FUNCTION_BLOCK FB_Infeed
VAR_INPUT
	bEnable_Master			: BOOL;
	bMoveMaster				: BOOL;
	bSensorProduct			: BOOL;
END_VAR

VAR_IN_OUT
	Master					: Axis_Ref;
	VirtMaster				: ARRAY [*] OF Axis_Ref;
END_VAR

VAR
	i						: DINT;
	iStartIndex				: DINT;
	VeloMaster				: LREAL;
	bToggle					: BOOL;

	fbPowerMaster			: MC_Power;
	fbMoveMaster			: MC_MoveVelocity;
	fbStopMaster			: MC_Halt;
	fbPowerVirtMaster		: ARRAY [1..iMaxNumbVirtMasters] OF MC_Power;
	fbVirtMaster			: ARRAY [1..iMaxNumbVirtMasters] OF FB_VirtualMaster;

END_VAR

// Enable Master
Master.ReadStatus();
fbPowerMaster(
	Axis			:= Master, 
	Enable			:= bEnable_Master, 
	Enable_Positive	:= bEnable_Master, 
	Enable_Negative	:= bEnable_Master, 
	Override		:= 100, 
	);
	
FOR i := 1 TO UPPER_BOUND(VirtMaster,1) DO
	VirtMaster[i].ReadStatus();
	fbPowerVirtMaster[i](
		Axis			:= VirtMaster[i], 
		Enable			:= bEnable_Master, 
		Enable_Positive	:= bEnable_Master, 
		Enable_Negative	:= bEnable_Master, 
		Override		:= 100, 
		);
END_FOR


// Start-Stop Master

VeloMaster := GVL_Infeed.iProductsPerMinute * 360 / 60;
bToggle:=NOT bToggle;

fbMoveMaster(
	Axis		:= Master, 
	Execute		:= bMoveMaster AND bToggle, 
	Velocity	:= VeloMaster, 
	Direction	:= MC_Positive_Direction, 
	);
fbStopMaster(
	Axis		:= Master, 
	Execute		:= NOT bMoveMaster, 
	);

// Virtual Master ready to start
iStartIndex:=0;
FOR i := 1 TO UPPER_BOUND(VirtMaster,1) DO
	IF VirtMaster[i].NcToPlc.ActPos=0 THEN
		iStartIndex:=i;
		i:=5;
	END_IF
END_FOR
	
// Detection product
FOR i := 1 TO UPPER_BOUND(VirtMaster,1) DO
	fbVirtMaster[i].bActivateCam:=FALSE;
END_FOR

IF (Master.NcToPlc.ModuloActPos > GVL_Infeed.rDetectionPosMin) AND (Master.NcToPlc.ModuloActPos < GVL_Infeed.rDetectionPosMax) AND bSensorProduct THEN
	fbVirtMaster[iStartIndex].bActivateCam:=TRUE;
END_IF
 
FOR i := 1 TO UPPER_BOUND(VirtMaster,1) DO
	fbVirtMaster[i](
		Master:= Master, 
		Slave:= VirtMaster[i],
		);
END_FOR

END_FUNCTION_BLOCK

(* stored: Version 1.1.0.1, ProductVersion 3.1.4024.12
   POU FB_Infeed: Id {10b295ba-01be-45b5-9e7a-224a70369683}, SpecialFunc None *)
